// TIA Portal V17 export
// export: Created 2025-03-05T08:03:41.9690947Z, ExportSetting WithDefaults, DisplayName Totally Integrated Automation Portal, DisplayVersion V17 Update 8, DisplayName TIA Portal Openness, DisplayVersion V17 Update 8, DisplayName TIA Portal Version Control Interface, DisplayVersion V17, DisplayName SINAMICS Startdrive Advanced, DisplayVersion V17 SP2, DisplayName SINAMICS Startdrive G110M, G120, G120C, G120D, G120P, G115D, DisplayVersion V17 SP2, DisplayName SINAMICS Startdrive G130, G150, S120, S150, SINAMICS MV, S210, DisplayVersion V17 SP2, DisplayName STEP 7 Professional, DisplayVersion V17 Update 8, DisplayName SINUMERIK ONE STEP 7 Toolbox, DisplayVersion V17 Update 12, DisplayName SINUMERIK 840D sl STEP 7 Toolbox, DisplayVersion V17 Update 12, DisplayName STEP 7 Safety, DisplayVersion V17 Update 6, DisplayName WinCC Advanced, DisplayVersion V17 Update 8
TYPE "POWDER FEEDER HOPPER"
// stored: IsFailsafeCompliant false
   STRUCT
      START_GENERAL_CONDITIONS : Bool;   // START GENERAL CONDITIONS
      START_INITIAL_CONDITIONS_LINE_1 : Bool;   // START INITIAL CONDITIONS LINE 1
      START_MANUAL_REQUEST_LINE_1 : Bool;   // START MANUAL REQUEST LINE 1
      START_INITIAL_CONDITIONS_LINE_2 : Bool;   // START INITIAL CONDITIONS LINE 2
      START_MANUAL_REQUEST_LINE_2 : Bool;   // START MANUAL REQUEST LINE 2
      START_AUTO_REQUEST : Bool;   // START AUTO REQUEST
      START_GLOBAL_REQUEST_LINE_1 : Bool;   // START GLOBAL REQUEST LINE 1
      START_COMMAND_LINE_1 : Bool;   // START COMMAND LINE 1
      START_LINE_1 : Bool;   // START LINE 1
      FEEDBACK_ON_LINE_1 : Bool;   // FEEDBACK ON LINE 1
      START_GLOBAL_REQUEST_LINE_2 : Bool;   // START GLOBAL REQUEST LINE 2
      START_COMMAND_LINE_2 : Bool;   // START COMMAND LINE 2
      START_LINE_2 : Bool;   // START LINE 2
      FEEDBACK_ON_LINE_2 : Bool;   // FEEDBACK ON LINE 2
      STOP_GENERAL_CONDITIONS : Bool;   // STOP GENERAL CONDITIONS
      STOP_INITIAL_CONDITIONS_LINE_1 : Bool;   // STOP INITIAL CONDITIONS LINE 1
      STOP_MANUAL_REQUEST_LINE_1 : Bool;   // STOP MANUAL REQUEST LINE 1
      STOP_INITIAL_CONDITIONS_LINE_2 : Bool;   // STOP INITIAL CONDITIONS LINE 2
      STOP_MANUAL_REQUEST_LINE_2 : Bool;   // STOP MANUAL REQUEST LINE 2
      STOP_AUTO_REQUEST : Bool;   // STOP AUTO REQUEST
      STOP_GLOBAL_REQUEST_LINE_1 : Bool;   // STOP GLOBAL REQUEST LINE 1
      STOP_COMMAND_LINE_1 : Bool;   // STOP COMMAND LINE 1
      STOP_LINE_1 : Bool;   // STOP LINE 1
      FEEDBACK_OFF_LINE_1 : Bool;   // FEEDBACK OFF LINE 1
      STOP_GLOBAL_REQUEST_LINE_2 : Bool;   // STOP GLOBAL REQUEST LINE 2
      STOP_COMMAND_LINE_2 : Bool;   // STOP COMMAND LINE 2
      STOP_LINE_2 : Bool;   // STOP LINE 2
      FEEDBACK_OFF_LINE_2 : Bool;   // FEEDBACK OFF LINE 2
      START_GENERAL_CONDITIONS_HELP : Bool;   // START GENERAL CONDITIONS HELP
      START_INITIAL_CONDITIONS_HELP : Bool;   // START INITIAL CONDITIONS HELP
      STOP_GENERAL_CONDITIONS_HELP : Bool;   // STOP GENERAL CONDITIONS HELP
      STOP_INITIAL_CONDITIONS_HELP : Bool;   // STOP INITIAL CONDITIONS HELP
      FAULT : Bool;   // FAULT
   END_STRUCT;
END_TYPE
